TYPE MoverComRequest :
STRUCT
  Start : BOOL;
  Stop : BOOL;
  GoHome : BOOL;
  Halt : BOOL;
END_STRUCT
END_TYPE

(* stored: Version 1.1.0.1
   DUT MoverComRequest: Id {926aa363-3fc6-4797-9e61-51f1f1d3bed3} *)
